DEVICE_TYPE RMT_DEV2 (* Subclass of RMT_DEV *)
  (* Standard: 61499-2 *)
  (* Version 0.0, 2005-03-26, JHC, Rockwell Automation *)
  (* Compiler header: package fb.rt.test;import fb.rt.ita.*; import fb.rt.math.*; *)
  (* Compiler classdef: public class RMT_DEV2 extends RMT_DEV *)
  RESOURCE RES1 : EMB_RES
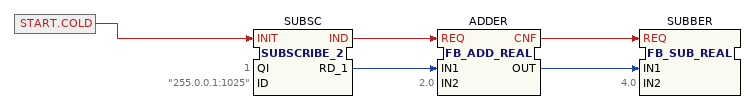
    FBS
      ADDER : FB_ADD_REAL(IN2 := 2.0);
      SUBBER : FB_SUB_REAL(IN2 := 4.0);
      SUBSC : SUBSCRIBE_2(QI := 1, ID := "255.0.0.1:1025");
    END_FBS
    EVENT_CONNECTIONS
      ADDER.CNF TO SUBBER.REQ;
      START.COLD TO SUBSC.INIT;
      SUBSC.IND TO ADDER.REQ;
    END_CONNECTIONS
    DATA_CONNECTIONS
      ADDER.OUT TO SUBBER.IN1;
      SUBSC.RD_1 TO ADDER.IN1;
    END_CONNECTIONS
  END_RESOURCE
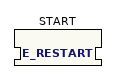
  FBS
    START : E_RESTART;
  END_FBS
END_DEVICE_TYPE
